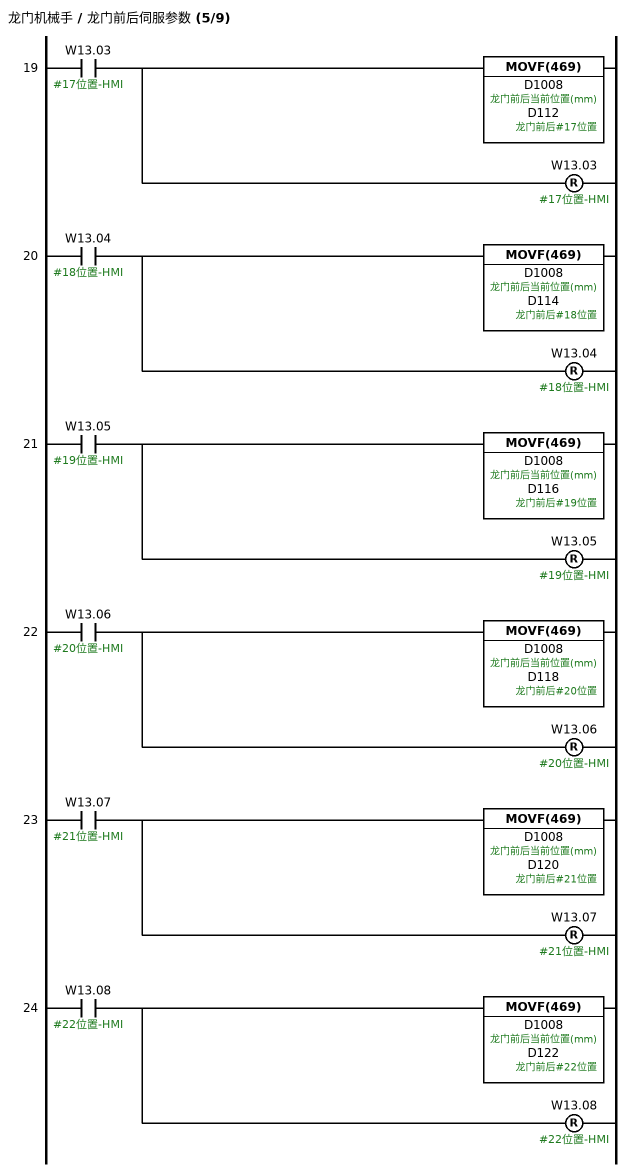
; [picture p305: 龙门机械手 / 龙门前后伺服参数, rungs 19-24]
; rung 19
LD W13.03  ; #17位置-HMI
MOVF(469) D1008 D112  ; 龙门前后当前位置(mm), 龙门前后#17位置
RSET W13.03  ; #17位置-HMI
; rung 20
LD W13.04  ; #18位置-HMI
MOVF(469) D1008 D114  ; 龙门前后当前位置(mm), 龙门前后#18位置
RSET W13.04  ; #18位置-HMI
; rung 21
LD W13.05  ; #19位置-HMI
MOVF(469) D1008 D116  ; 龙门前后当前位置(mm), 龙门前后#19位置
RSET W13.05  ; #19位置-HMI
; rung 22
LD W13.06  ; #20位置-HMI
MOVF(469) D1008 D118  ; 龙门前后当前位置(mm), 龙门前后#20位置
RSET W13.06  ; #20位置-HMI
; rung 23
LD W13.07  ; #21位置-HMI
MOVF(469) D1008 D120  ; 龙门前后当前位置(mm), 龙门前后#21位置
RSET W13.07  ; #21位置-HMI
; rung 24
LD W13.08  ; #22位置-HMI
MOVF(469) D1008 D122  ; 龙门前后当前位置(mm), 龙门前后#22位置
RSET W13.08  ; #22位置-HMI

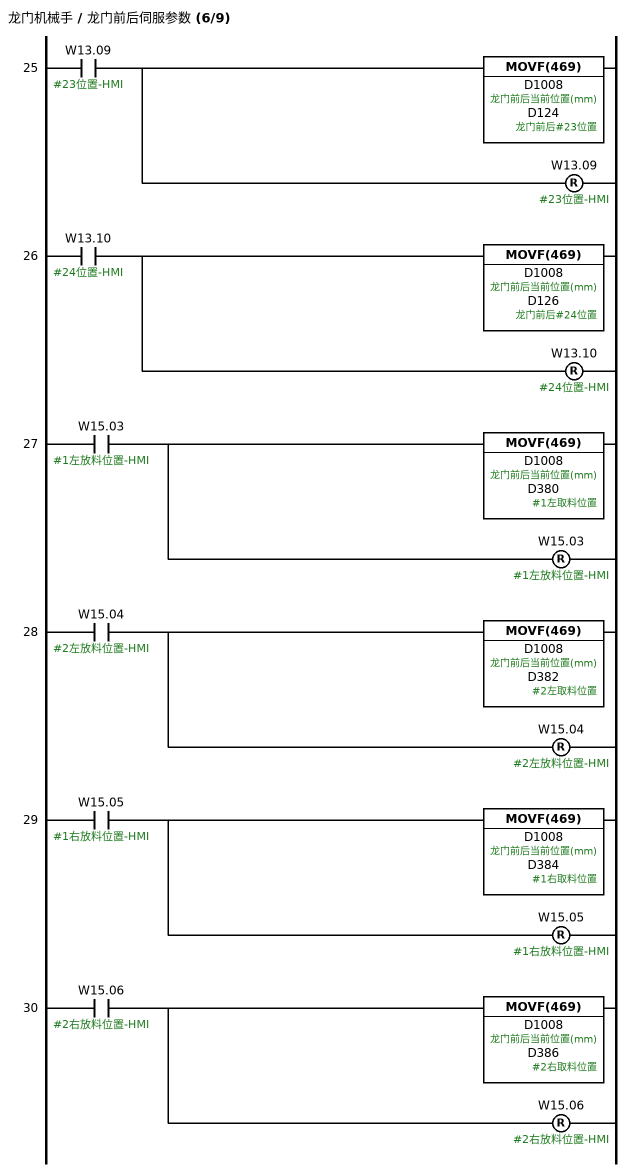
; rung 25
LD W13.09  ; #23位置-HMI
MOVF(469) D1008 D124  ; 龙门前后当前位置(mm), 龙门前后#23位置
RSET W13.09  ; #23位置-HMI
; rung 26
LD W13.10  ; #24位置-HMI
MOVF(469) D1008 D126  ; 龙门前后当前位置(mm), 龙门前后#24位置
RSET W13.10  ; #24位置-HMI
; rung 27
LD W15.03  ; #1左放料位置-HMI
MOVF(469) D1008 D380  ; 龙门前后当前位置(mm), #1左取料位置
RSET W15.03  ; #1左放料位置-HMI
; rung 28
LD W15.04  ; #2左放料位置-HMI
MOVF(469) D1008 D382  ; 龙门前后当前位置(mm), #2左取料位置
RSET W15.04  ; #2左放料位置-HMI
; rung 29
LD W15.05  ; #1右放料位置-HMI
MOVF(469) D1008 D384  ; 龙门前后当前位置(mm), #1右取料位置
RSET W15.05  ; #1右放料位置-HMI
; rung 30
LD W15.06  ; #2右放料位置-HMI
MOVF(469) D1008 D386  ; 龙门前后当前位置(mm), #2右取料位置
RSET W15.06  ; #2右放料位置-HMI

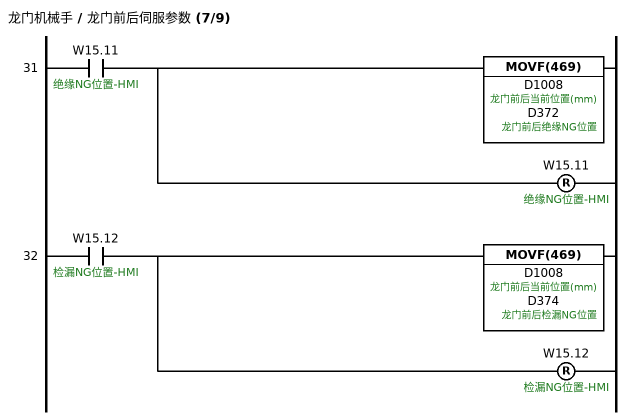
; rung 31
LD W15.11  ; 绝缘NG位置-HMI
MOVF(469) D1008 D372  ; 龙门前后当前位置(mm), 龙门前后绝缘NG位置
RSET W15.11  ; 绝缘NG位置-HMI
; rung 32
LD W15.12  ; 检漏NG位置-HMI
MOVF(469) D1008 D374  ; 龙门前后当前位置(mm), 龙门前后检漏NG位置
RSET W15.12  ; 检漏NG位置-HMI

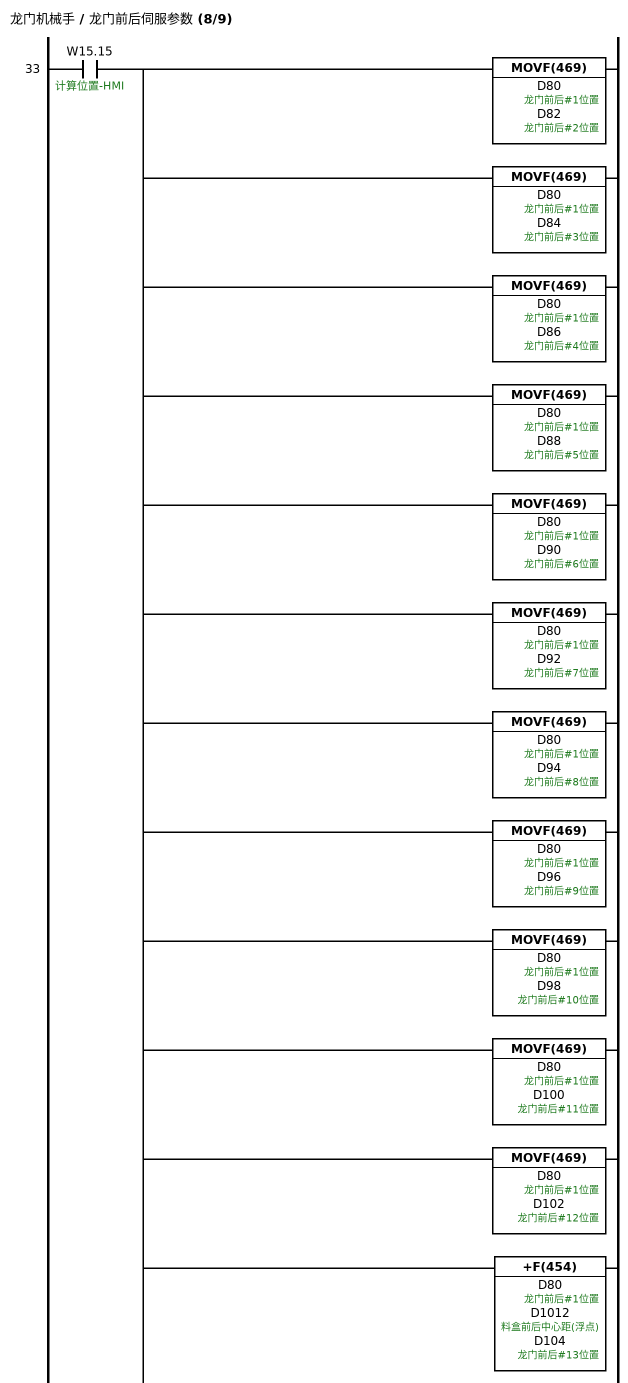

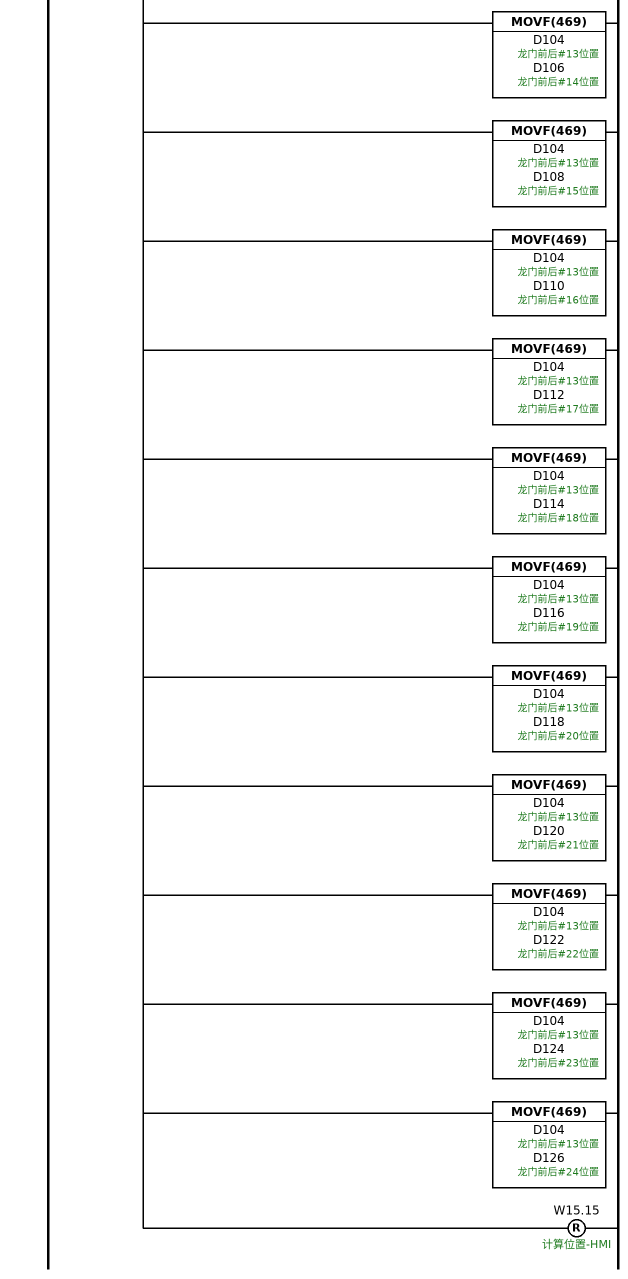
; rung 33
LD W15.15  ; 计算位置-HMI
MOVF(469) D80 D82  ; 龙门前后#1位置, 龙门前后#2位置
MOVF(469) D80 D84  ; 龙门前后#1位置, 龙门前后#3位置
MOVF(469) D80 D86  ; 龙门前后#1位置, 龙门前后#4位置
MOVF(469) D80 D88  ; 龙门前后#1位置, 龙门前后#5位置
MOVF(469) D80 D90  ; 龙门前后#1位置, 龙门前后#6位置
MOVF(469) D80 D92  ; 龙门前后#1位置, 龙门前后#7位置
MOVF(469) D80 D94  ; 龙门前后#1位置, 龙门前后#8位置
MOVF(469) D80 D96  ; 龙门前后#1位置, 龙门前后#9位置
MOVF(469) D80 D98  ; 龙门前后#1位置, 龙门前后#10位置
MOVF(469) D80 D100  ; 龙门前后#1位置, 龙门前后#11位置
MOVF(469) D80 D102  ; 龙门前后#1位置, 龙门前后#12位置
+F(454) D80 D1012 D104  ; 龙门前后#1位置, 料盒前后中心距(浮点), 龙门前后#13位置
MOVF(469) D104 D106  ; 龙门前后#13位置, 龙门前后#14位置
MOVF(469) D104 D108  ; 龙门前后#13位置, 龙门前后#15位置
MOVF(469) D104 D110  ; 龙门前后#13位置, 龙门前后#16位置
MOVF(469) D104 D112  ; 龙门前后#13位置, 龙门前后#17位置
MOVF(469) D104 D114  ; 龙门前后#13位置, 龙门前后#18位置
MOVF(469) D104 D116  ; 龙门前后#13位置, 龙门前后#19位置
MOVF(469) D104 D118  ; 龙门前后#13位置, 龙门前后#20位置
MOVF(469) D104 D120  ; 龙门前后#13位置, 龙门前后#21位置
MOVF(469) D104 D122  ; 龙门前后#13位置, 龙门前后#22位置
MOVF(469) D104 D124  ; 龙门前后#13位置, 龙门前后#23位置
MOVF(469) D104 D126  ; 龙门前后#13位置, 龙门前后#24位置
RSET W15.15  ; 计算位置-HMI

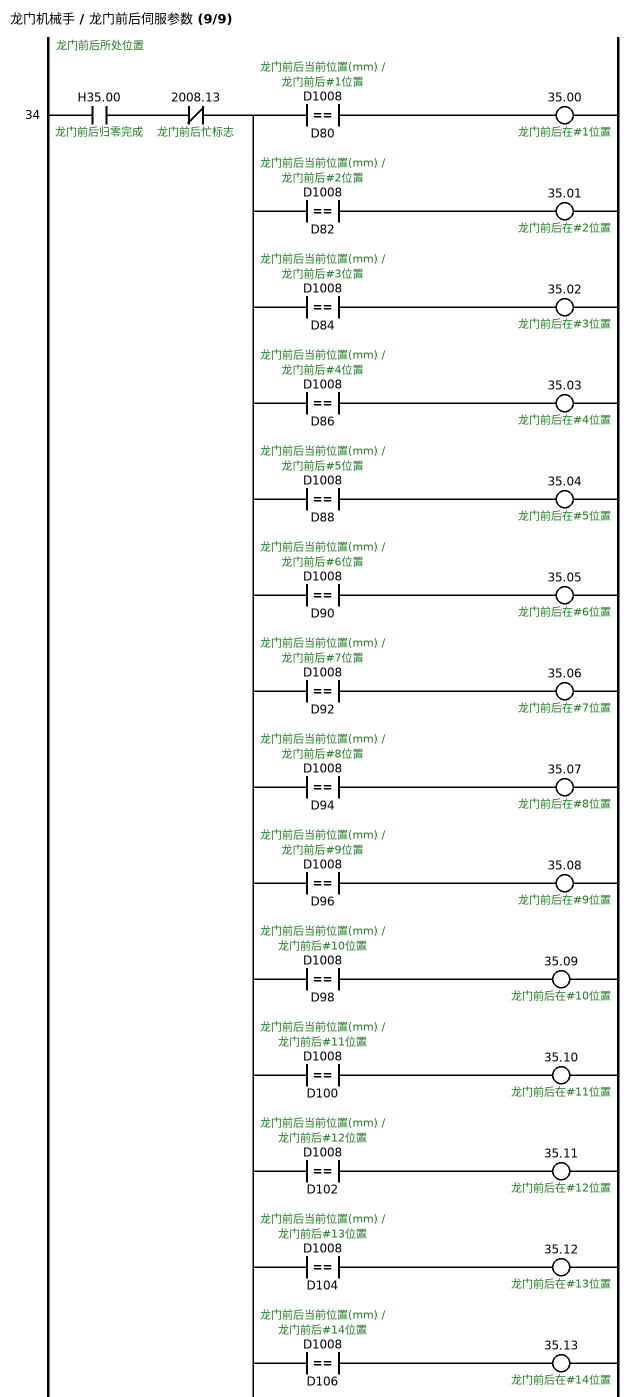

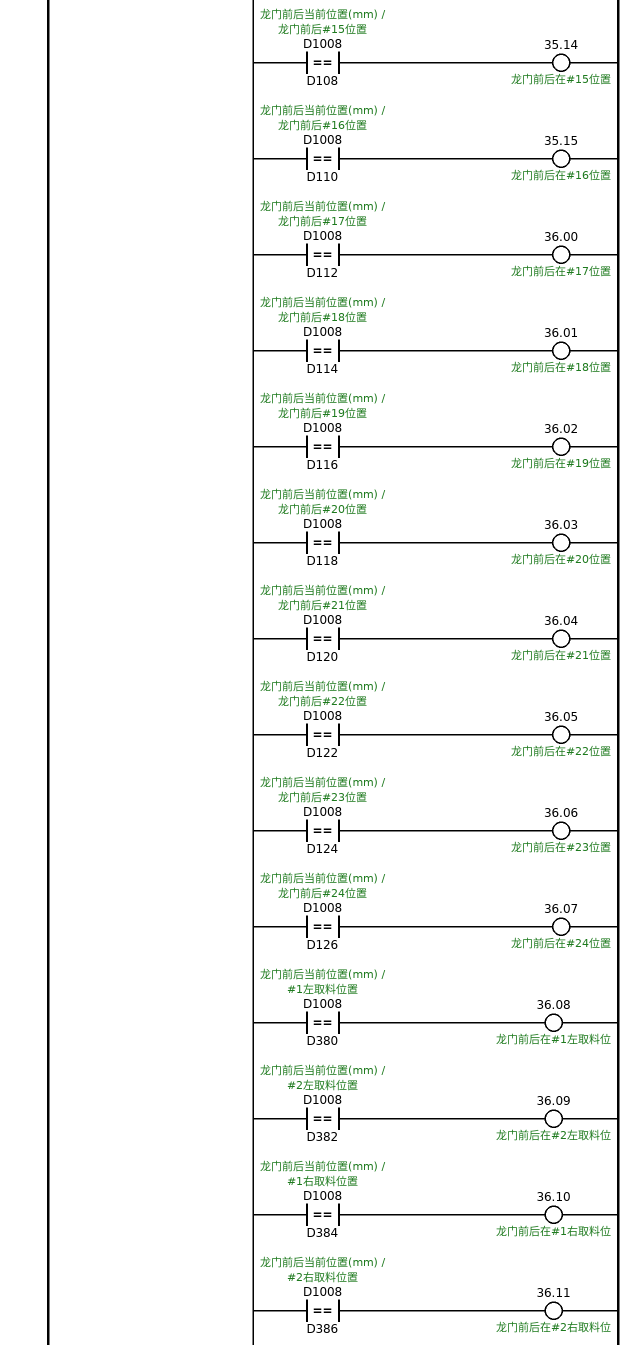

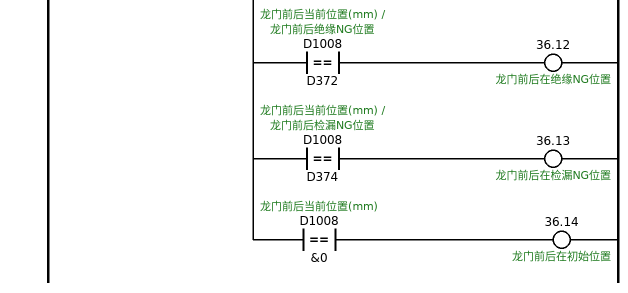
; rung 34: 龙门前后所处位置
LD H35.00  ; 龙门前后归零完成
ANDNOT 2008.13  ; 龙门前后忙标志
OUT TR0
AND=F(329) D1008 D80  ; 龙门前后当前位置(mm), 龙门前后#1位置
OUT 35.00  ; 龙门前后在#1位置
LD TR0
AND=F(329) D1008 D82  ; 龙门前后当前位置(mm), 龙门前后#2位置
OUT 35.01  ; 龙门前后在#2位置
LD TR0
AND=F(329) D1008 D84  ; 龙门前后当前位置(mm), 龙门前后#3位置
OUT 35.02  ; 龙门前后在#3位置
LD TR0
AND=F(329) D1008 D86  ; 龙门前后当前位置(mm), 龙门前后#4位置
OUT 35.03  ; 龙门前后在#4位置
LD TR0
AND=F(329) D1008 D88  ; 龙门前后当前位置(mm), 龙门前后#5位置
OUT 35.04  ; 龙门前后在#5位置
LD TR0
AND=F(329) D1008 D90  ; 龙门前后当前位置(mm), 龙门前后#6位置
OUT 35.05  ; 龙门前后在#6位置
LD TR0
AND=F(329) D1008 D92  ; 龙门前后当前位置(mm), 龙门前后#7位置
OUT 35.06  ; 龙门前后在#7位置
LD TR0
AND=F(329) D1008 D94  ; 龙门前后当前位置(mm), 龙门前后#8位置
OUT 35.07  ; 龙门前后在#8位置
LD TR0
AND=F(329) D1008 D96  ; 龙门前后当前位置(mm), 龙门前后#9位置
OUT 35.08  ; 龙门前后在#9位置
LD TR0
AND=F(329) D1008 D98  ; 龙门前后当前位置(mm), 龙门前后#10位置
OUT 35.09  ; 龙门前后在#10位置
LD TR0
AND=F(329) D1008 D100  ; 龙门前后当前位置(mm), 龙门前后#11位置
OUT 35.10  ; 龙门前后在#11位置
LD TR0
AND=F(329) D1008 D102  ; 龙门前后当前位置(mm), 龙门前后#12位置
OUT 35.11  ; 龙门前后在#12位置
LD TR0
AND=F(329) D1008 D104  ; 龙门前后当前位置(mm), 龙门前后#13位置
OUT 35.12  ; 龙门前后在#13位置
LD TR0
AND=F(329) D1008 D106  ; 龙门前后当前位置(mm), 龙门前后#14位置
OUT 35.13  ; 龙门前后在#14位置
LD TR0
AND=F(329) D1008 D108  ; 龙门前后当前位置(mm), 龙门前后#15位置
OUT 35.14  ; 龙门前后在#15位置
LD TR0
AND=F(329) D1008 D110  ; 龙门前后当前位置(mm), 龙门前后#16位置
OUT 35.15  ; 龙门前后在#16位置
LD TR0
AND=F(329) D1008 D112  ; 龙门前后当前位置(mm), 龙门前后#17位置
OUT 36.00  ; 龙门前后在#17位置
LD TR0
AND=F(329) D1008 D114  ; 龙门前后当前位置(mm), 龙门前后#18位置
OUT 36.01  ; 龙门前后在#18位置
LD TR0
AND=F(329) D1008 D116  ; 龙门前后当前位置(mm), 龙门前后#19位置
OUT 36.02  ; 龙门前后在#19位置
LD TR0
AND=F(329) D1008 D118  ; 龙门前后当前位置(mm), 龙门前后#20位置
OUT 36.03  ; 龙门前后在#20位置
LD TR0
AND=F(329) D1008 D120  ; 龙门前后当前位置(mm), 龙门前后#21位置
OUT 36.04  ; 龙门前后在#21位置
LD TR0
AND=F(329) D1008 D122  ; 龙门前后当前位置(mm), 龙门前后#22位置
OUT 36.05  ; 龙门前后在#22位置
LD TR0
AND=F(329) D1008 D124  ; 龙门前后当前位置(mm), 龙门前后#23位置
OUT 36.06  ; 龙门前后在#23位置
LD TR0
AND=F(329) D1008 D126  ; 龙门前后当前位置(mm), 龙门前后#24位置
OUT 36.07  ; 龙门前后在#24位置
LD TR0
AND=F(329) D1008 D380  ; 龙门前后当前位置(mm), #1左取料位置
OUT 36.08  ; 龙门前后在#1左取料位
LD TR0
AND=F(329) D1008 D382  ; 龙门前后当前位置(mm), #2左取料位置
OUT 36.09  ; 龙门前后在#2左取料位
LD TR0
AND=F(329) D1008 D384  ; 龙门前后当前位置(mm), #1右取料位置
OUT 36.10  ; 龙门前后在#1右取料位
LD TR0
AND=F(329) D1008 D386  ; 龙门前后当前位置(mm), #2右取料位置
OUT 36.11  ; 龙门前后在#2右取料位
LD TR0
AND=F(329) D1008 D372  ; 龙门前后当前位置(mm), 龙门前后绝缘NG位置
OUT 36.12  ; 龙门前后在绝缘NG位置
LD TR0
AND=F(329) D1008 D374  ; 龙门前后当前位置(mm), 龙门前后检漏NG位置
OUT 36.13  ; 龙门前后在检漏NG位置
LD TR0
AND=F(329) D1008 &0  ; 龙门前后当前位置(mm)
OUT 36.14  ; 龙门前后在初始位置

### Section 龙门左右伺服参数

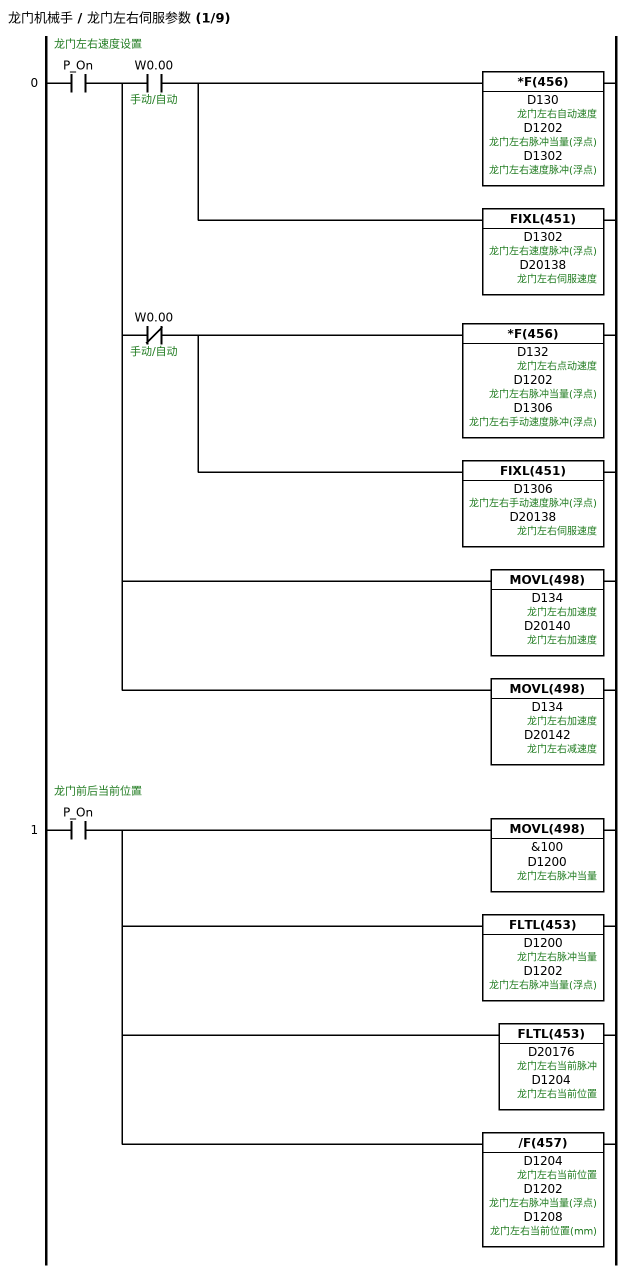
; rung 0: 龙门左右速度设置
LD P_On
OUT TR0
AND W0.00  ; 手动/自动
*F(456) D130 D1202 D1302  ; 龙门左右自动速度, 龙门左右脉冲当量(浮点), 龙门左右速度脉冲(浮点)
FIXL(451) D1302 D20138  ; 龙门左右速度脉冲(浮点), 龙门左右伺服速度
LD TR0
ANDNOT W0.00  ; 手动/自动
*F(456) D132 D1202 D1306  ; 龙门左右点动速度, 龙门左右脉冲当量(浮点), 龙门左右手动速度脉冲(浮点)
FIXL(451) D1306 D20138  ; 龙门左右手动速度脉冲(浮点), 龙门左右伺服速度
LD TR0
MOVL(498) D134 D20140  ; 龙门左右加速度
MOVL(498) D134 D20142  ; 龙门左右加速度, 龙门左右减速度
; rung 1: 龙门前后当前位置
LD P_On
MOVL(498) &100 D1200  ; 龙门左右脉冲当量
FLTL(453) D1200 D1202  ; 龙门左右脉冲当量, 龙门左右脉冲当量(浮点)
FLTL(453) D20176 D1204  ; 龙门左右当前脉冲, 龙门左右当前位置
/F(457) D1204 D1202 D1208  ; 龙门左右当前位置, 龙门左右脉冲当量(浮点), 龙门左右当前位置(mm)

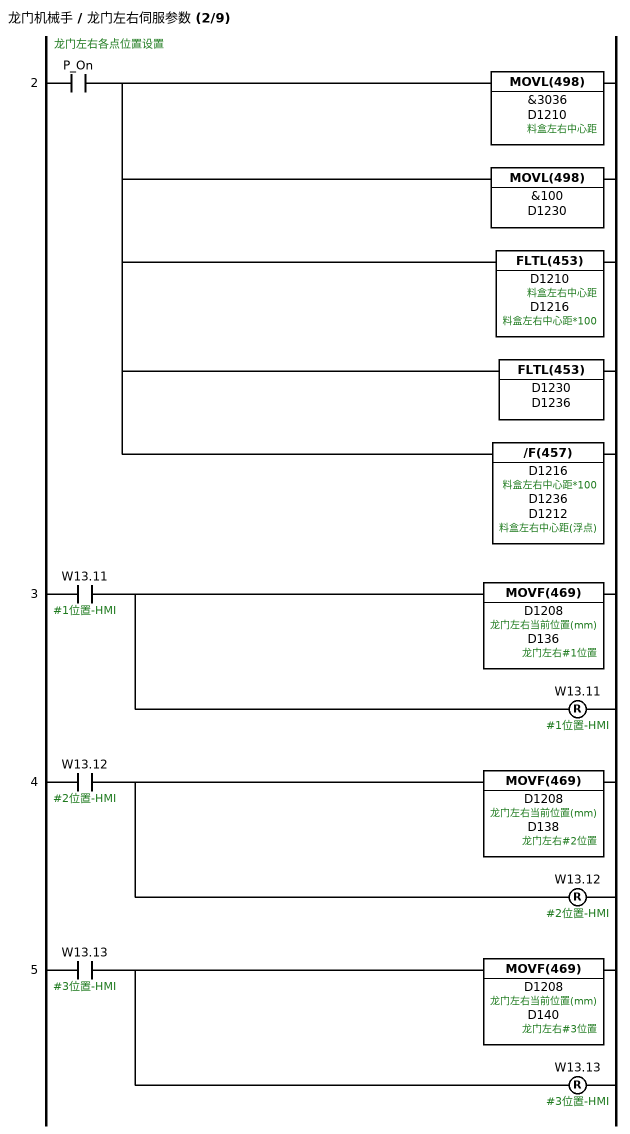
; rung 2: 龙门左右各点位置设置
LD P_On
MOVL(498) &3036 D1210  ; 料盒左右中心距
MOVL(498) &100 D1230
FLTL(453) D1210 D1216  ; 料盒左右中心距, 料盒左右中心距*100
FLTL(453) D1230 D1236
/F(457) D1216 D1236 D1212  ; 料盒左右中心距*100, 料盒左右中心距(浮点)
; rung 3
LD W13.11  ; #1位置-HMI
MOVF(469) D1208 D136  ; 龙门左右当前位置(mm), 龙门左右#1位置
RSET W13.11  ; #1位置-HMI
; rung 4
LD W13.12  ; #2位置-HMI
MOVF(469) D1208 D138  ; 龙门左右当前位置(mm), 龙门左右#2位置
RSET W13.12  ; #2位置-HMI
; rung 5
LD W13.13  ; #3位置-HMI
MOVF(469) D1208 D140  ; 龙门左右当前位置(mm), 龙门左右#3位置
RSET W13.13  ; #3位置-HMI

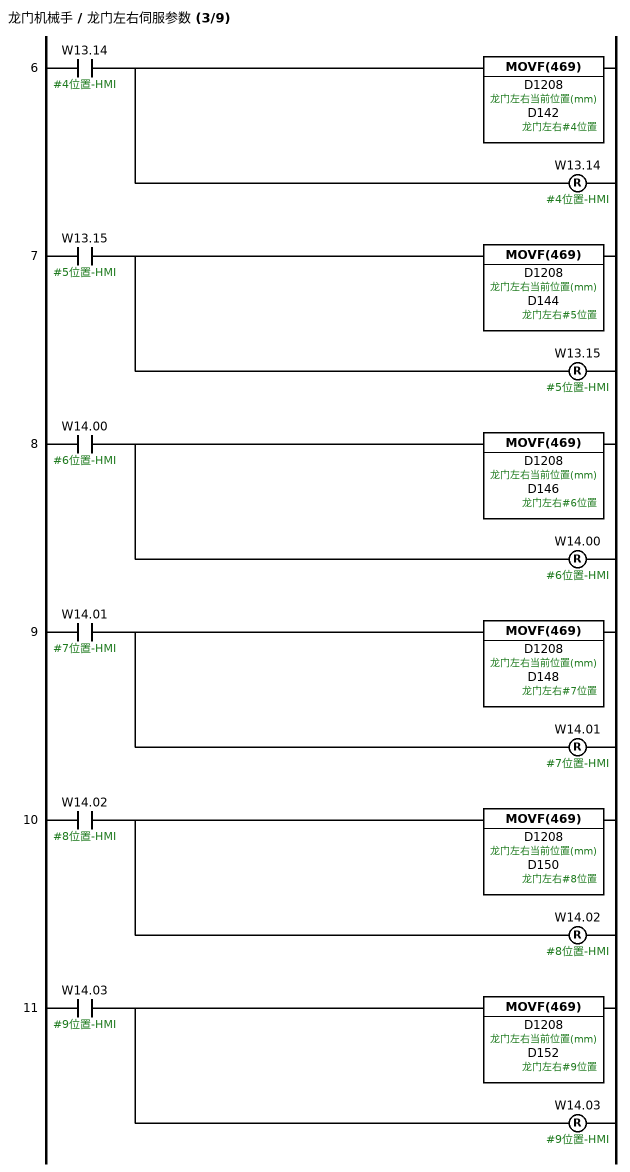
; rung 6
LD W13.14  ; #4位置-HMI
MOVF(469) D1208 D142  ; 龙门左右当前位置(mm), 龙门左右#4位置
RSET W13.14  ; #4位置-HMI
; rung 7
LD W13.15  ; #5位置-HMI
MOVF(469) D1208 D144  ; 龙门左右当前位置(mm), 龙门左右#5位置
RSET W13.15  ; #5位置-HMI
; rung 8
LD W14.00  ; #6位置-HMI
MOVF(469) D1208 D146  ; 龙门左右当前位置(mm), 龙门左右#6位置
RSET W14.00  ; #6位置-HMI
; rung 9
LD W14.01  ; #7位置-HMI
MOVF(469) D1208 D148  ; 龙门左右当前位置(mm), 龙门左右#7位置
RSET W14.01  ; #7位置-HMI
; rung 10
LD W14.02  ; #8位置-HMI
MOVF(469) D1208 D150  ; 龙门左右当前位置(mm), 龙门左右#8位置
RSET W14.02  ; #8位置-HMI
; rung 11
LD W14.03  ; #9位置-HMI
MOVF(469) D1208 D152  ; 龙门左右当前位置(mm), 龙门左右#9位置
RSET W14.03  ; #9位置-HMI

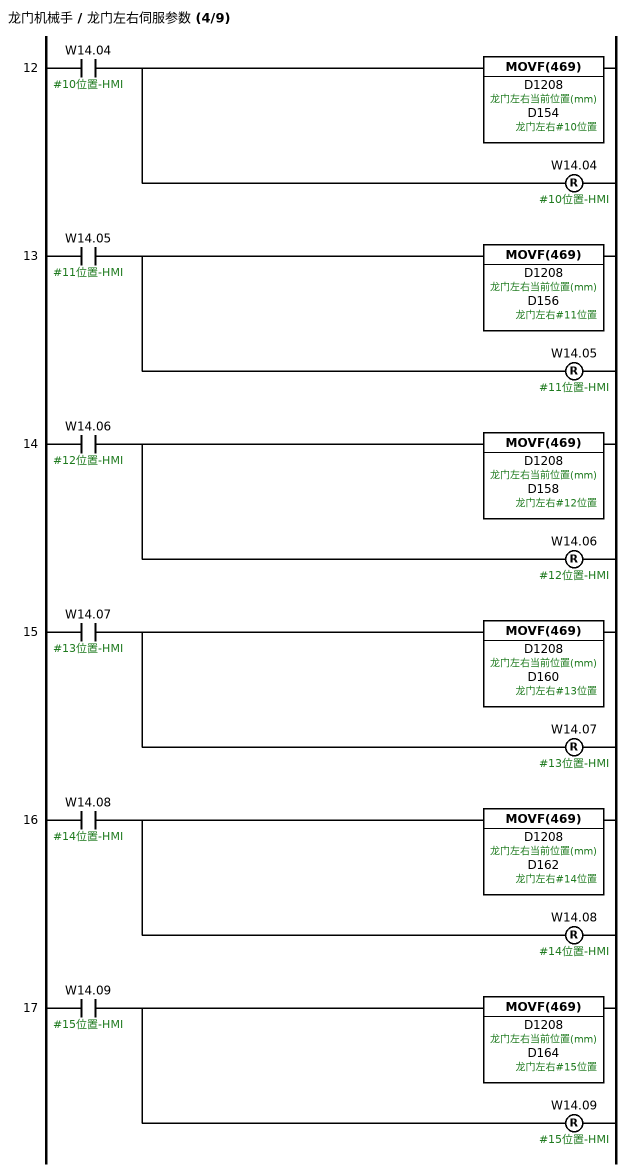
; rung 12
LD W14.04  ; #10位置-HMI
MOVF(469) D1208 D154  ; 龙门左右当前位置(mm), 龙门左右#10位置
RSET W14.04  ; #10位置-HMI
; rung 13
LD W14.05  ; #11位置-HMI
MOVF(469) D1208 D156  ; 龙门左右当前位置(mm), 龙门左右#11位置
RSET W14.05  ; #11位置-HMI
; rung 14
LD W14.06  ; #12位置-HMI
MOVF(469) D1208 D158  ; 龙门左右当前位置(mm), 龙门左右#12位置
RSET W14.06  ; #12位置-HMI
; rung 15
LD W14.07  ; #13位置-HMI
MOVF(469) D1208 D160  ; 龙门左右当前位置(mm), 龙门左右#13位置
RSET W14.07  ; #13位置-HMI
; rung 16
LD W14.08  ; #14位置-HMI
MOVF(469) D1208 D162  ; 龙门左右当前位置(mm), 龙门左右#14位置
RSET W14.08  ; #14位置-HMI
; rung 17
LD W14.09  ; #15位置-HMI
MOVF(469) D1208 D164  ; 龙门左右当前位置(mm), 龙门左右#15位置
RSET W14.09  ; #15位置-HMI

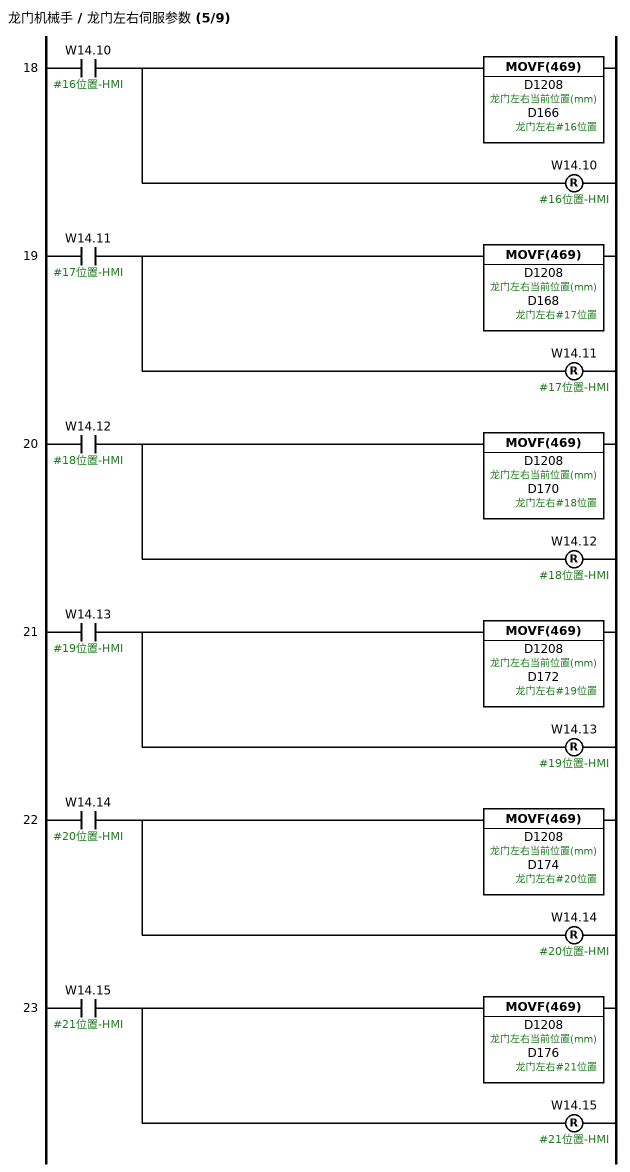
; rung 18
LD W14.10  ; #16位置-HMI
MOVF(469) D1208 D166  ; 龙门左右当前位置(mm), 龙门左右#16位置
RSET W14.10  ; #16位置-HMI
; rung 19
LD W14.11  ; #17位置-HMI
MOVF(469) D1208 D168  ; 龙门左右当前位置(mm), 龙门左右#17位置
RSET W14.11  ; #17位置-HMI
; rung 20
LD W14.12  ; #18位置-HMI
MOVF(469) D1208 D170  ; 龙门左右当前位置(mm), 龙门左右#18位置
RSET W14.12  ; #18位置-HMI
; rung 21
LD W14.13  ; #19位置-HMI
MOVF(469) D1208 D172  ; 龙门左右当前位置(mm), 龙门左右#19位置
RSET W14.13  ; #19位置-HMI
; rung 22
LD W14.14  ; #20位置-HMI
MOVF(469) D1208 D174  ; 龙门左右当前位置(mm), 龙门左右#20位置
RSET W14.14  ; #20位置-HMI
; rung 23
LD W14.15  ; #21位置-HMI
MOVF(469) D1208 D176  ; 龙门左右当前位置(mm), 龙门左右#21位置
RSET W14.15  ; #21位置-HMI

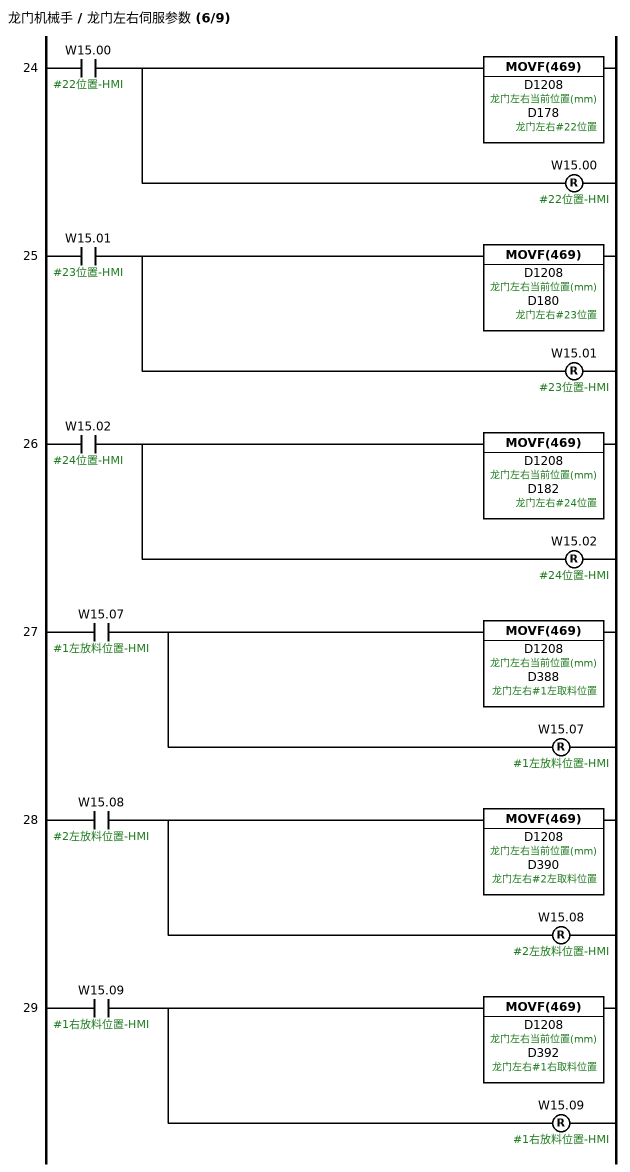
; rung 24
LD W15.00  ; #22位置-HMI
MOVF(469) D1208 D178  ; 龙门左右当前位置(mm), 龙门左右#22位置
RSET W15.00  ; #22位置-HMI
; rung 25
LD W15.01  ; #23位置-HMI
MOVF(469) D1208 D180  ; 龙门左右当前位置(mm), 龙门左右#23位置
RSET W15.01  ; #23位置-HMI
; rung 26
LD W15.02  ; #24位置-HMI
MOVF(469) D1208 D182  ; 龙门左右当前位置(mm), 龙门左右#24位置
RSET W15.02  ; #24位置-HMI
; rung 27
LD W15.07  ; #1左放料位置-HMI
MOVF(469) D1208 D388  ; 龙门左右当前位置(mm), 龙门左右#1左取料位置
RSET W15.07  ; #1左放料位置-HMI
; rung 28
LD W15.08  ; #2左放料位置-HMI
MOVF(469) D1208 D390  ; 龙门左右当前位置(mm), 龙门左右#2左取料位置
RSET W15.08  ; #2左放料位置-HMI
; rung 29
LD W15.09  ; #1右放料位置-HMI
MOVF(469) D1208 D392  ; 龙门左右当前位置(mm), 龙门左右#1右取料位置
RSET W15.09  ; #1右放料位置-HMI

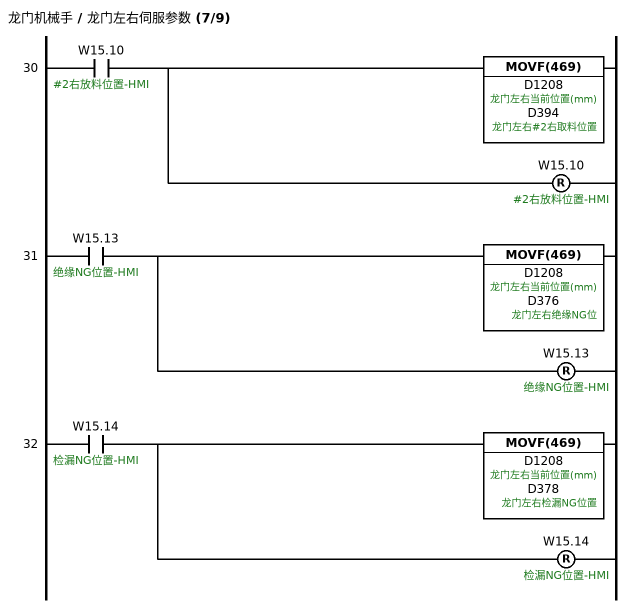
; rung 30
LD W15.10  ; #2右放料位置-HMI
MOVF(469) D1208 D394  ; 龙门左右当前位置(mm), 龙门左右#2右取料位置
RSET W15.10  ; #2右放料位置-HMI
; rung 31
LD W15.13  ; 绝缘NG位置-HMI
MOVF(469) D1208 D376  ; 龙门左右当前位置(mm), 龙门左右绝缘NG位
RSET W15.13  ; 绝缘NG位置-HMI
; rung 32
LD W15.14  ; 检漏NG位置-HMI
MOVF(469) D1208 D378  ; 龙门左右当前位置(mm), 龙门左右检漏NG位置
RSET W15.14  ; 检漏NG位置-HMI

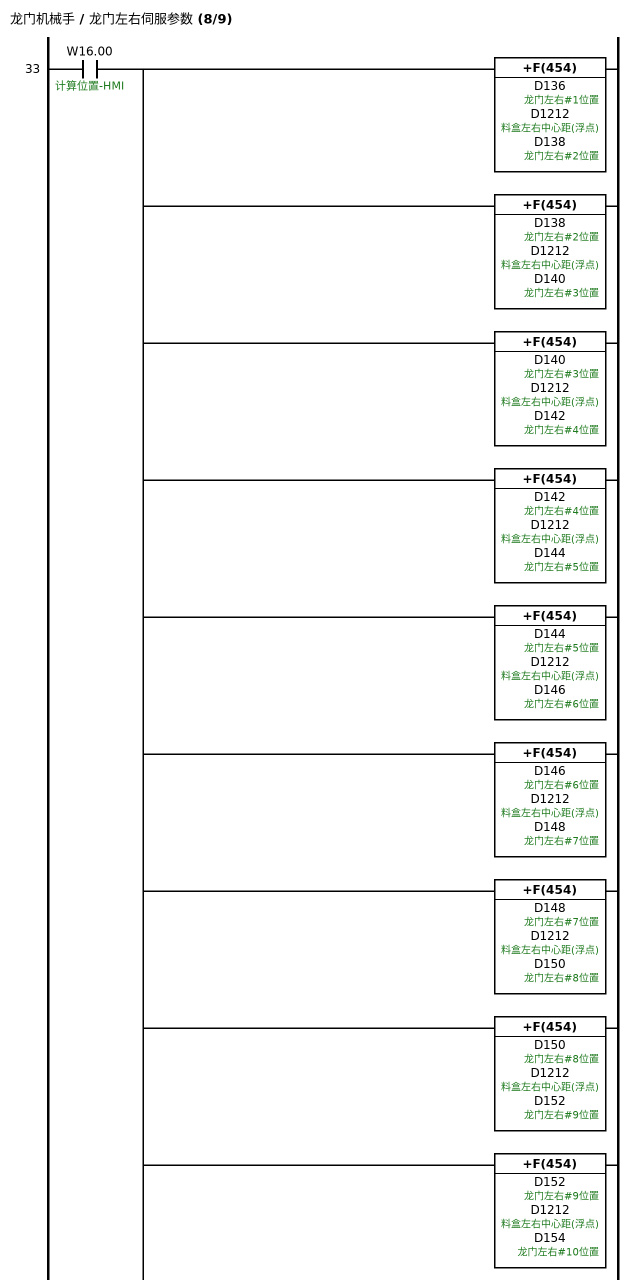

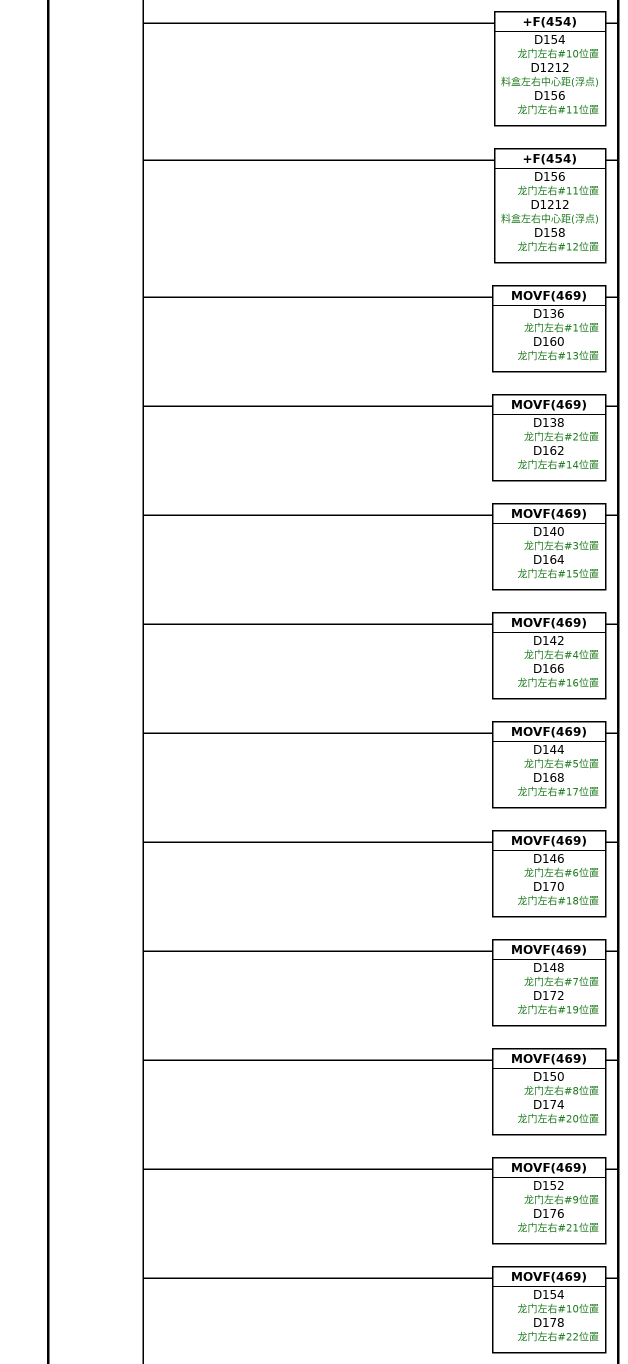

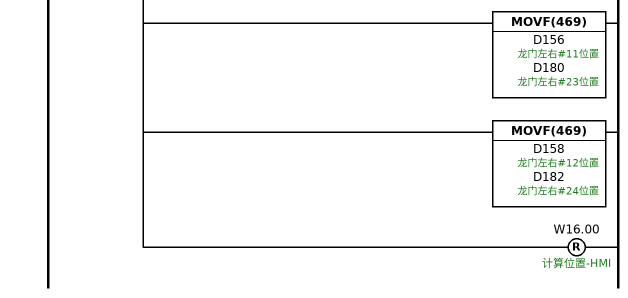
; rung 33
LD W16.00  ; 计算位置-HMI
+F(454) D136 D1212 D138  ; 龙门左右#1位置, 料盒左右中心距(浮点), 龙门左右#2位置
+F(454) D138 D1212 D140  ; 龙门左右#2位置, 料盒左右中心距(浮点), 龙门左右#3位置
+F(454) D140 D1212 D142  ; 龙门左右#3位置, 料盒左右中心距(浮点), 龙门左右#4位置
+F(454) D142 D1212 D144  ; 龙门左右#4位置, 料盒左右中心距(浮点), 龙门左右#5位置
+F(454) D144 D1212 D146  ; 龙门左右#5位置, 料盒左右中心距(浮点), 龙门左右#6位置
+F(454) D146 D1212 D148  ; 龙门左右#6位置, 料盒左右中心距(浮点), 龙门左右#7位置
+F(454) D148 D1212 D150  ; 龙门左右#7位置, 料盒左右中心距(浮点), 龙门左右#8位置
+F(454) D150 D1212 D152  ; 龙门左右#8位置, 料盒左右中心距(浮点), 龙门左右#9位置
+F(454) D152 D1212 D154  ; 龙门左右#9位置, 料盒左右中心距(浮点), 龙门左右#10位置
+F(454) D154 D1212 D156  ; 龙门左右#10位置, 料盒左右中心距(浮点), 龙门左右#11位置
+F(454) D156 D1212 D158  ; 龙门左右#11位置, 料盒左右中心距(浮点), 龙门左右#12位置
MOVF(469) D136 D160  ; 龙门左右#1位置, 龙门左右#13位置
MOVF(469) D138 D162  ; 龙门左右#2位置, 龙门左右#14位置
MOVF(469) D140 D164  ; 龙门左右#3位置, 龙门左右#15位置
MOVF(469) D142 D166  ; 龙门左右#4位置, 龙门左右#16位置
MOVF(469) D144 D168  ; 龙门左右#5位置, 龙门左右#17位置
MOVF(469) D146 D170  ; 龙门左右#6位置, 龙门左右#18位置
MOVF(469) D148 D172  ; 龙门左右#7位置, 龙门左右#19位置
MOVF(469) D150 D174  ; 龙门左右#8位置, 龙门左右#20位置
MOVF(469) D152 D176  ; 龙门左右#9位置, 龙门左右#21位置
MOVF(469) D154 D178  ; 龙门左右#10位置, 龙门左右#22位置
MOVF(469) D156 D180  ; 龙门左右#11位置, 龙门左右#23位置
MOVF(469) D158 D182  ; 龙门左右#12位置, 龙门左右#24位置
RSET W16.00  ; 计算位置-HMI

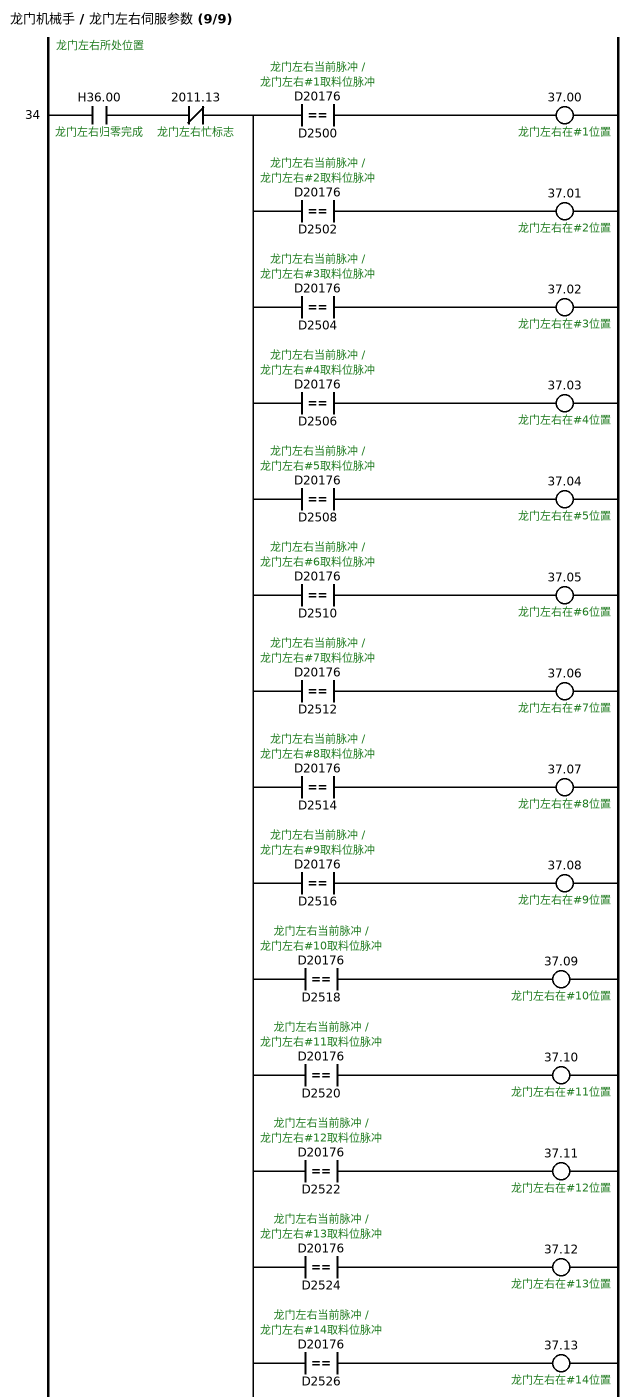

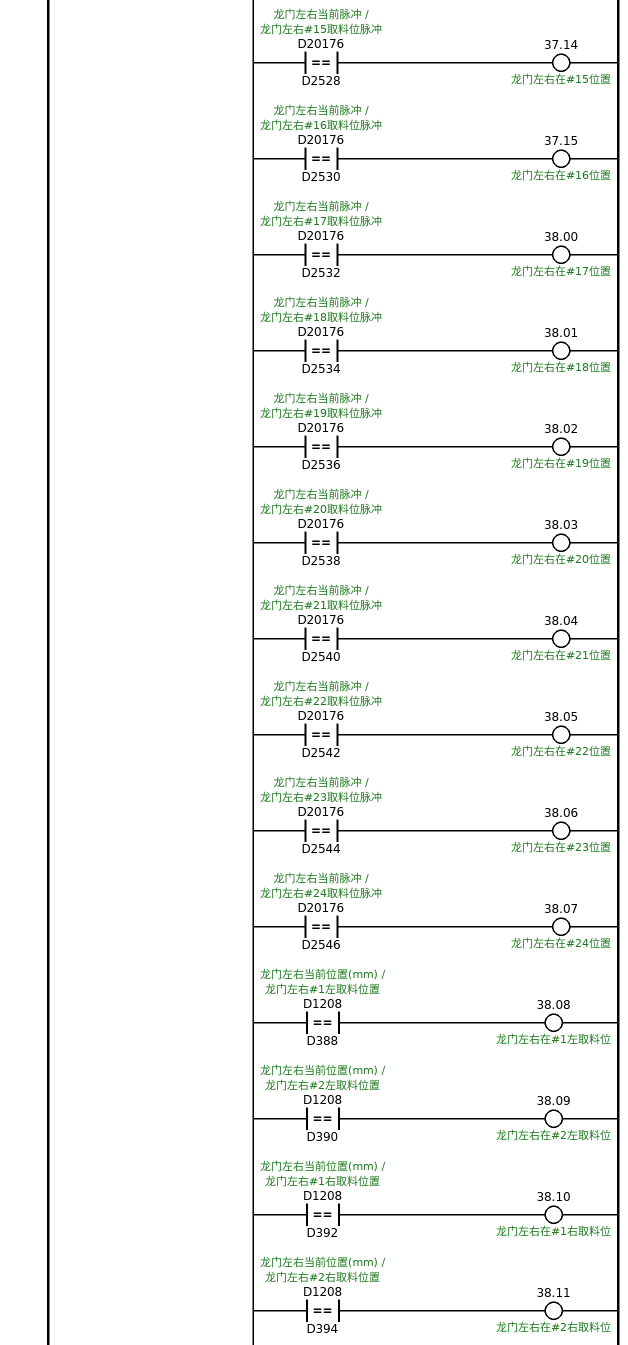

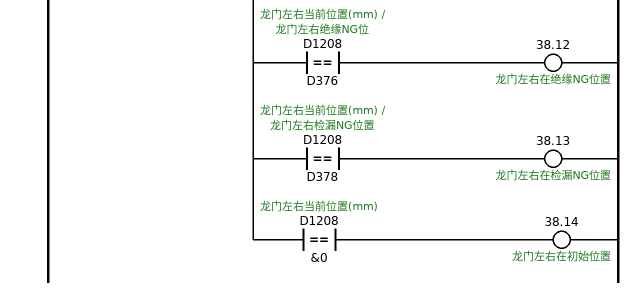
; rung 34: 龙门左右所处位置
LD H36.00  ; 龙门左右归零完成
ANDNOT 2011.13  ; 龙门左右忙标志
OUT TR0
AND=(300) D20176 D2500  ; 龙门左右当前脉冲, 龙门左右#1取料位脉冲
OUT 37.00  ; 龙门左右在#1位置
LD TR0
AND=(300) D20176 D2502  ; 龙门左右当前脉冲, 龙门左右#2取料位脉冲
OUT 37.01  ; 龙门左右在#2位置
LD TR0
AND=(300) D20176 D2504  ; 龙门左右当前脉冲, 龙门左右#3取料位脉冲
OUT 37.02  ; 龙门左右在#3位置
LD TR0
AND=(300) D20176 D2506  ; 龙门左右当前脉冲, 龙门左右#4取料位脉冲
OUT 37.03  ; 龙门左右在#4位置
LD TR0
AND=(300) D20176 D2508  ; 龙门左右当前脉冲, 龙门左右#5取料位脉冲
OUT 37.04  ; 龙门左右在#5位置
LD TR0
AND=(300) D20176 D2510  ; 龙门左右当前脉冲, 龙门左右#6取料位脉冲
OUT 37.05  ; 龙门左右在#6位置
LD TR0
AND=(300) D20176 D2512  ; 龙门左右当前脉冲, 龙门左右#7取料位脉冲
OUT 37.06  ; 龙门左右在#7位置
LD TR0
AND=(300) D20176 D2514  ; 龙门左右当前脉冲, 龙门左右#8取料位脉冲
OUT 37.07  ; 龙门左右在#8位置
LD TR0
AND=(300) D20176 D2516  ; 龙门左右当前脉冲, 龙门左右#9取料位脉冲
OUT 37.08  ; 龙门左右在#9位置
LD TR0
AND=(300) D20176 D2518  ; 龙门左右当前脉冲, 龙门左右#10取料位脉冲
OUT 37.09  ; 龙门左右在#10位置
LD TR0
AND=(300) D20176 D2520  ; 龙门左右当前脉冲, 龙门左右#11取料位脉冲
OUT 37.10  ; 龙门左右在#11位置
LD TR0
AND=(300) D20176 D2522  ; 龙门左右当前脉冲, 龙门左右#12取料位脉冲
OUT 37.11  ; 龙门左右在#12位置
LD TR0
AND=(300) D20176 D2524  ; 龙门左右当前脉冲, 龙门左右#13取料位脉冲
OUT 37.12  ; 龙门左右在#13位置
LD TR0
AND=(300) D20176 D2526  ; 龙门左右当前脉冲, 龙门左右#14取料位脉冲
OUT 37.13  ; 龙门左右在#14位置
LD TR0
AND=(300) D20176 D2528  ; 龙门左右当前脉冲, 龙门左右#15取料位脉冲
OUT 37.14  ; 龙门左右在#15位置
LD TR0
AND=(300) D20176 D2530  ; 龙门左右当前脉冲, 龙门左右#16取料位脉冲
OUT 37.15  ; 龙门左右在#16位置
LD TR0
AND=(300) D20176 D2532  ; 龙门左右当前脉冲, 龙门左右#17取料位脉冲
OUT 38.00  ; 龙门左右在#17位置
LD TR0
AND=(300) D20176 D2534  ; 龙门左右当前脉冲, 龙门左右#18取料位脉冲
OUT 38.01  ; 龙门左右在#18位置
LD TR0
AND=(300) D20176 D2536  ; 龙门左右当前脉冲, 龙门左右#19取料位脉冲
OUT 38.02  ; 龙门左右在#19位置
LD TR0
AND=(300) D20176 D2538  ; 龙门左右当前脉冲, 龙门左右#20取料位脉冲
OUT 38.03  ; 龙门左右在#20位置
LD TR0
AND=(300) D20176 D2540  ; 龙门左右当前脉冲, 龙门左右#21取料位脉冲
OUT 38.04  ; 龙门左右在#21位置
LD TR0
AND=(300) D20176 D2542  ; 龙门左右当前脉冲, 龙门左右#22取料位脉冲
OUT 38.05  ; 龙门左右在#22位置
LD TR0
AND=(300) D20176 D2544  ; 龙门左右当前脉冲, 龙门左右#23取料位脉冲
OUT 38.06  ; 龙门左右在#23位置
LD TR0
AND=(300) D20176 D2546  ; 龙门左右当前脉冲, 龙门左右#24取料位脉冲
OUT 38.07  ; 龙门左右在#24位置
LD TR0
AND=F(329) D1208 D388  ; 龙门左右当前位置(mm), 龙门左右#1左取料位置
OUT 38.08  ; 龙门左右在#1左取料位
LD TR0
AND=F(329) D1208 D390  ; 龙门左右当前位置(mm), 龙门左右#2左取料位置
OUT 38.09  ; 龙门左右在#2左取料位
LD TR0
AND=F(329) D1208 D392  ; 龙门左右当前位置(mm), 龙门左右#1右取料位置
OUT 38.10  ; 龙门左右在#1右取料位
LD TR0
AND=F(329) D1208 D394  ; 龙门左右当前位置(mm), 龙门左右#2右取料位置
OUT 38.11  ; 龙门左右在#2右取料位
LD TR0
AND=F(329) D1208 D376  ; 龙门左右当前位置(mm), 龙门左右绝缘NG位
OUT 38.12  ; 龙门左右在绝缘NG位置
LD TR0
AND=F(329) D1208 D378  ; 龙门左右当前位置(mm), 龙门左右检漏NG位置
OUT 38.13  ; 龙门左右在检漏NG位置
LD TR0
AND=F(329) D1208 &0  ; 龙门左右当前位置(mm)
OUT 38.14  ; 龙门左右在初始位置

### Section 料盒升降伺服参数

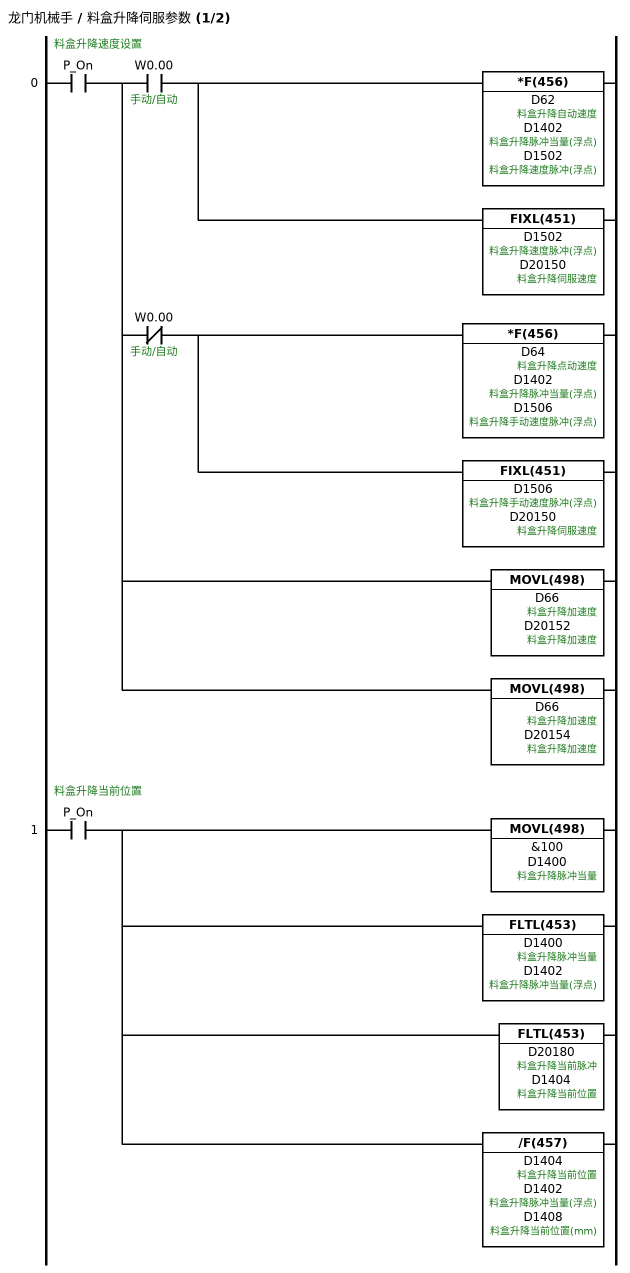
; rung 0: 料盒升降速度设置
LD P_On
OUT TR0
AND W0.00  ; 手动/自动
*F(456) D62 D1402 D1502  ; 料盒升降自动速度, 料盒升降脉冲当量(浮点), 料盒升降速度脉冲(浮点)
FIXL(451) D1502 D20150  ; 料盒升降速度脉冲(浮点), 料盒升降伺服速度
LD TR0
ANDNOT W0.00  ; 手动/自动
*F(456) D64 D1402 D1506  ; 料盒升降点动速度, 料盒升降脉冲当量(浮点), 料盒升降手动速度脉冲(浮点)
FIXL(451) D1506 D20150  ; 料盒升降手动速度脉冲(浮点), 料盒升降伺服速度
LD TR0
MOVL(498) D66 D20152  ; 料盒升降加速度
MOVL(498) D66 D20154  ; 料盒升降加速度
; rung 1: 料盒升降当前位置
LD P_On
MOVL(498) &100 D1400  ; 料盒升降脉冲当量
FLTL(453) D1400 D1402  ; 料盒升降脉冲当量, 料盒升降脉冲当量(浮点)
FLTL(453) D20180 D1404  ; 料盒升降当前脉冲, 料盒升降当前位置
/F(457) D1404 D1402 D1408  ; 料盒升降当前位置, 料盒升降脉冲当量(浮点), 料盒升降当前位置(mm)

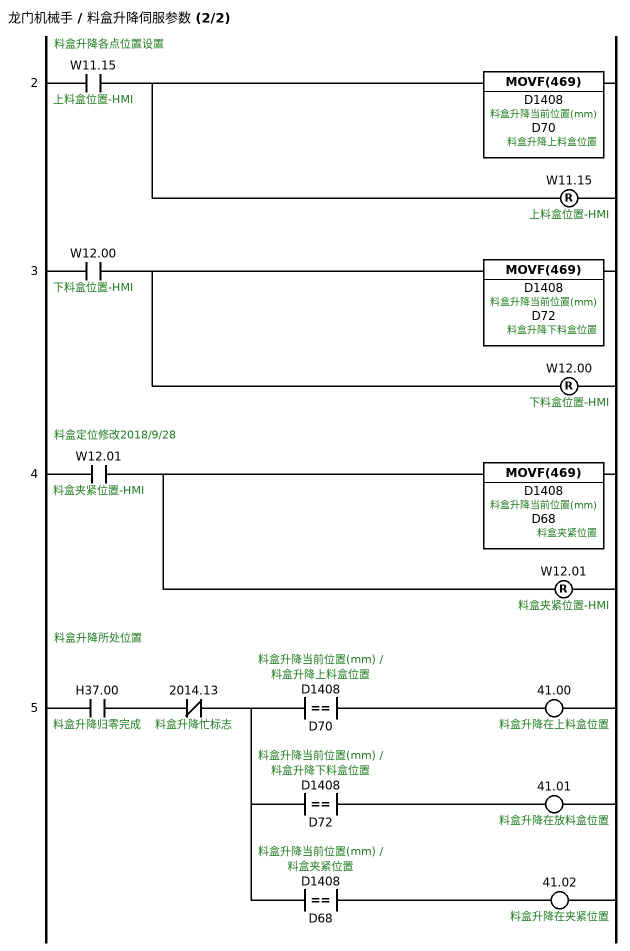
; rung 2: 料盒升降各点位置设置
LD W11.15  ; 上料盒位置-HMI
MOVF(469) D1408 D70  ; 料盒升降当前位置(mm), 料盒升降上料盒位置
RSET W11.15  ; 上料盒位置-HMI
; rung 3
LD W12.00  ; 下料盒位置-HMI
MOVF(469) D1408 D72  ; 料盒升降当前位置(mm), 料盒升降下料盒位置
RSET W12.00  ; 下料盒位置-HMI
; rung 4: 料盒定位修改2018/9/28
LD W12.01  ; 料盒夹紧位置-HMI
MOVF(469) D1408 D68  ; 料盒升降当前位置(mm), 料盒夹紧位置
RSET W12.01  ; 料盒夹紧位置-HMI
; rung 5: 料盒升降所处位置
LD H37.00  ; 料盒升降归零完成
ANDNOT 2014.13  ; 料盒升降忙标志
OUT TR0
AND=F(329) D1408 D70  ; 料盒升降当前位置(mm), 料盒升降上料盒位置
OUT 41.00  ; 料盒升降在上料盒位置
LD TR0
AND=F(329) D1408 D72  ; 料盒升降当前位置(mm), 料盒升降下料盒位置
OUT 41.01  ; 料盒升降在放料盒位置
LD TR0
AND=F(329) D1408 D68  ; 料盒升降当前位置(mm), 料盒夹紧位置
OUT 41.02  ; 料盒升降在夹紧位置

### Section 龙门前后、左右轴控输出

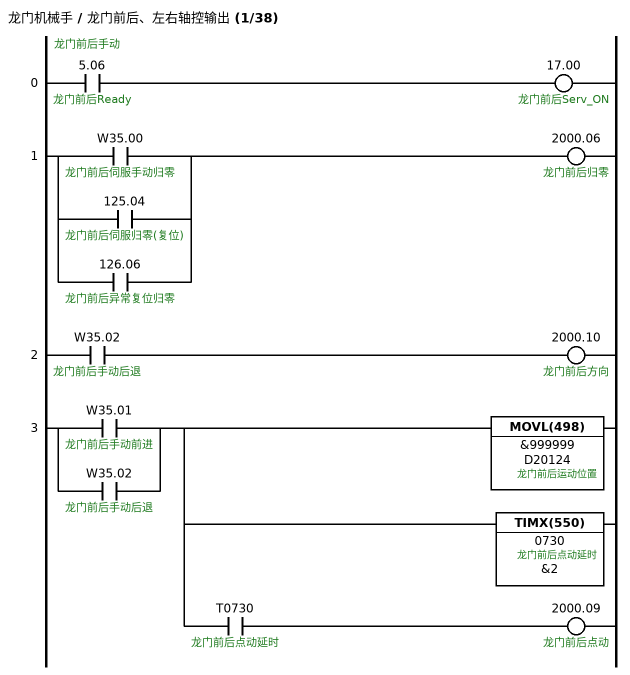
; rung 0: 龙门前后手动
LD 5.06  ; 龙门前后Ready
OUT 17.00  ; 龙门前后Serv_ON
; rung 1
LD W35.00  ; 龙门前后伺服手动归零
OR 125.04  ; 龙门前后伺服归零(复位)
OR 126.06  ; 龙门前后异常复位归零
OUT 2000.06  ; 龙门前后归零
; rung 2
LD W35.02  ; 龙门前后手动后退
OUT 2000.10  ; 龙门前后方向
; rung 3
LD W35.01  ; 龙门前后手动前进
OR W35.02  ; 龙门前后手动后退
MOVL(498) &999999 D20124  ; 龙门前后运动位置
TIMX(550) 0730 &2  ; 龙门前后点动延时
AND T0730  ; 龙门前后点动延时
OUT 2000.09  ; 龙门前后点动

